(* CODESYS project Übung1.project

Project tree, tasks and I/O mapping:
  CODESYS_Control_Win_V3_x64 : CODESYS Control Win V3, 3S - Smart Software Solutions GmbH, version 3.5.3.60
    application Application
      task VISU_TASK (cyclic, interval 100 ms, priority 30) calls VisuElems.Visu_Prg
      task MainTask (cyclic, interval t#20ms, priority 1) calls Alarmmeldung
      program Alarmmeldung [LD]
      visualisation Alarmmeldung_Vis
  text list GlobalTextList
*)

// CODESYS_Control_Win_V3_x64/Application/Alarmmeldung
PROGRAM Alarmmeldung
VAR
	S1: BOOL;
	S2: BOOL;
	S3: BOOL;
	Alarm: BOOL;
END_VAR

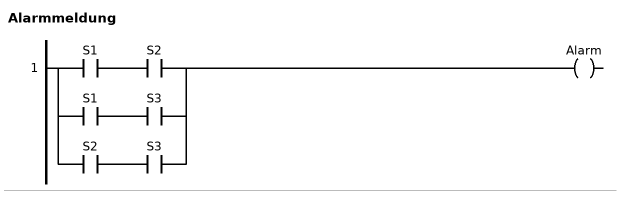
// NETWORK 1
Alarm := S1 AND S2 OR S1 AND S3 OR S2 AND S3;

END_PROGRAM

// CODESYS_Control_Win_V3_x64/Application/Alarmmeldung_Vis
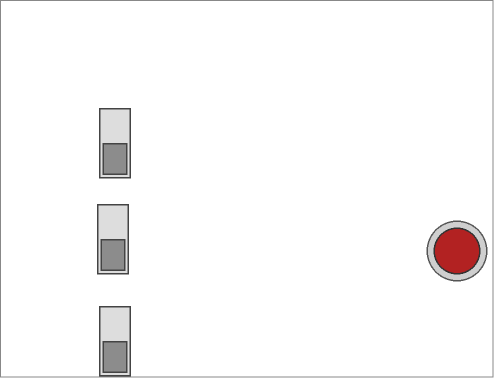
VISUALIZATION Alarmmeldung_Vis  // 494x378
    DipSwitch (80,108 70x70), tooltip "S1", variable: Alarmmeldung.S1, behaviour: TOGGLE, style: Switch-DipSwitch-Gray
    DipSwitch (78,204 70x70), tooltip "S2", variable: Alarmmeldung.S2, behaviour: TOGGLE, style: Switch-DipSwitch-Gray
    DipSwitch (80,306 70x70), tooltip "S3", variable: Alarmmeldung.S3, behaviour: TOGGLE, style: Switch-DipSwitch-Gray
    Lamp1 (422,216 70x70), tooltip "Alarm", variable: Alarmmeldung.Alarm, style: Lamp-Lamp1-Red
END_VISUALIZATION
